// TIA Portal V17 export
// export: Created 2023-04-11T09:33:28.1593293Z, ExportSetting WithDefaults, DisplayName Totally Integrated Automation Portal, DisplayVersion V17 Update 3, DisplayName TIA Portal Openness, DisplayVersion V17 Update 3, DisplayName TIA Portal Version Control Interface, DisplayVersion V17, DisplayName SINAMICS Startdrive Advanced, DisplayVersion V17 Update2, DisplayName SINAMICS Startdrive G130, G150, S120, S150, SINAMICS MV, S210, DisplayVersion V17 Update2, DisplayName SINAMICS Startdrive G110M, G120, G120C, G120D, G120P, G115D, DisplayVersion V17 Update2, DisplayName STEP 7 Professional, DisplayVersion V17 Update 3, DisplayName STEP 7 Safety, DisplayVersion V17, DisplayName WinCC UA Professional, DisplayVersion V17 Update 3
FUNCTION_BLOCK "FB_stdCylinder"   // FB121, LAD
TITLE = Standart cylinder control
{ S7_Optimized_Access := 'TRUE' }
VERSION : 0.1
// stored: AutoNumber true, IsIECCheckEnabled false, IsRetainMemResEnabled false, MemoryReserve 100, SetENOAutomatically false, UDAEnableTagReadback false
   VAR_INPUT
      Double_Coil : Bool;
      Request_A : Bool;
      Request_B : Bool;
      Sensor_A : Bool;
      With_A : Bool;
      Sensor_B : Bool;
      With_B : Bool;
      Enable_A : Bool;
      Enable_B : Bool;
      Monitoring_On : Bool;
      SensorDelay_A : Time;
      SensorDelay_B : Time;
      TimeForError_A : Time;
      TimeForError_B : Time;
   END_VAR
   VAR_OUTPUT
      Out_A : Bool;
      Out_B : Bool;
      Done_A : Bool;
      Done_B : Bool;
      Error_A : Bool;
      Error_B : Bool;
      Error_moveBlock : Bool;
   END_VAR
   VAR
      FB_FaultModule_Instance { S7_SetPoint := 'True'} : "FB_faultModule";
      IEC_Timer_0_Instance { S7_SetPoint := 'True'} : TON_TIME;
      IEC_Timer_0_Instance_1 { S7_SetPoint := 'True'} : TON_TIME;
      IEC_Timer_0_Instance_2 { S7_SetPoint := 'True'} : TON_TIME;
      IEC_Timer_0_Instance_3 { S7_SetPoint := 'True'} : TON_TIME;
   END_VAR
   VAR_TEMP
      Out_A_temp : Bool;
      Out_B_temp : Bool;
   END_VAR
BEGIN

REGION Network 1: OUT A
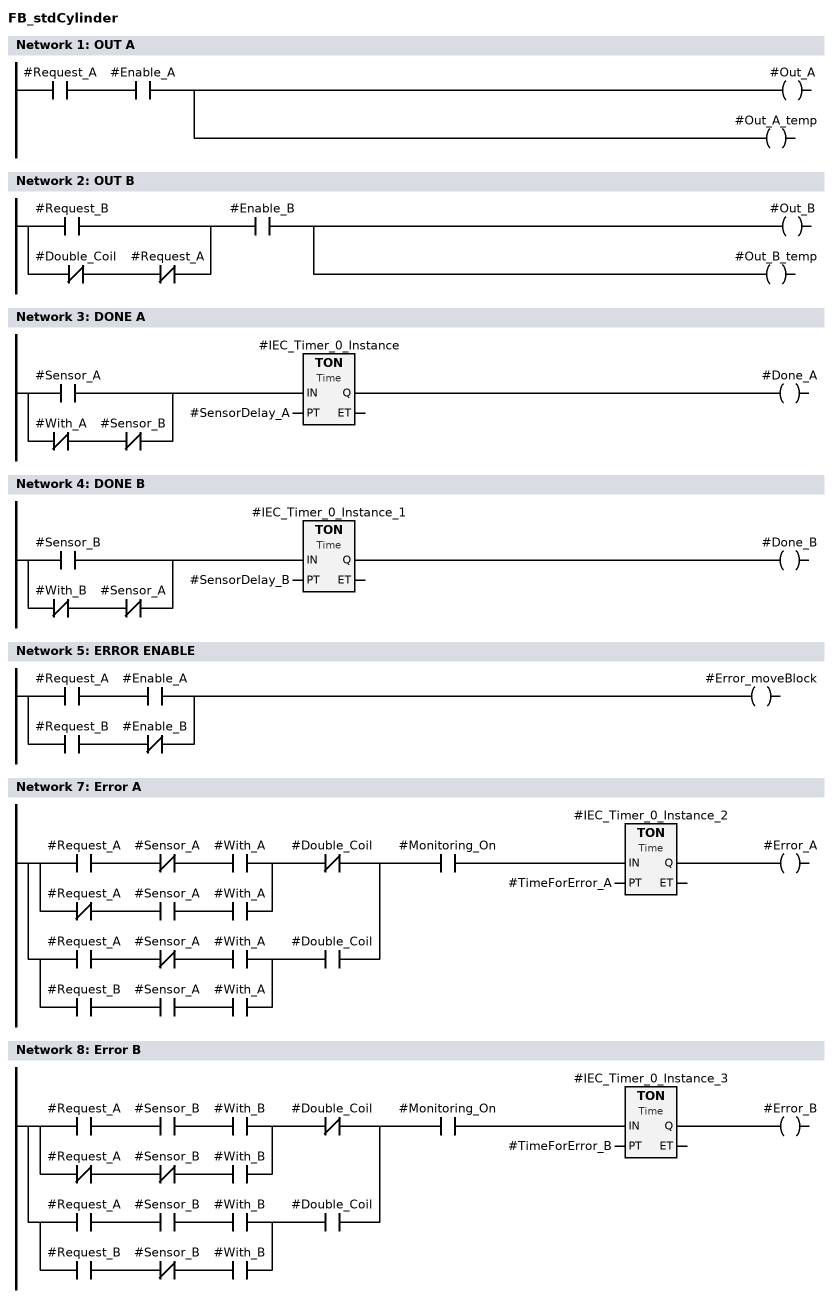
   RUNG wire#powerrail
      Contact( #Request_A )
      Contact( #Enable_A )
      wire#w1
      Coil( #Out_A )
   END_RUNG
   RUNG wire#w1
      Coil( #Out_A_temp )
   END_RUNG
   // the same network as SCL:
   #Out_A := #Request_A AND #Enable_A;
   #Out_A_temp := #Out_A;
END_REGION

REGION Network 2: OUT B
   RUNG wire#powerrail
      Contact( #Request_B )
      wire#w1
      Contact( #Enable_B )
      wire#w2
      Coil( #Out_B )
   END_RUNG
   RUNG wire#powerrail
      I_Contact( #Double_Coil )
      I_Contact( #Request_A )
   END_RUNG wire#w1
   RUNG wire#w2
      Coil( #Out_B_temp )
   END_RUNG
   // the same network as SCL:
   #Out_B := (#Request_B OR (NOT #Double_Coil AND NOT #Request_A)) AND #Enable_B;
   #Out_B_temp := #Out_B;
END_REGION

REGION Network 3: DONE A
   RUNG wire#powerrail
      Contact( #Sensor_A )
      wire#w1
      { S7_Templates := "time_type := Time" } #IEC_Timer_0_Instance.TON(pt := #SensorDelay_A, et =>)
      Coil( #Done_A )
   END_RUNG
   RUNG wire#powerrail
      I_Contact( #With_A )
      I_Contact( #Sensor_B )
   END_RUNG wire#w1
   // the same network as SCL:
   #IEC_Timer_0_Instance(IN := #Sensor_A OR (NOT #With_A AND NOT #Sensor_B), PT := #SensorDelay_A);   // TON
   #Done_A := #IEC_Timer_0_Instance.Q;
END_REGION

REGION Network 4: DONE B
   RUNG wire#powerrail
      Contact( #Sensor_B )
      wire#w1
      { S7_Templates := "time_type := Time" } #IEC_Timer_0_Instance_1.TON(pt := #SensorDelay_B, et =>)
      Coil( #Done_B )
   END_RUNG
   RUNG wire#powerrail
      I_Contact( #With_B )
      I_Contact( #Sensor_A )
   END_RUNG wire#w1
   // the same network as SCL:
   #IEC_Timer_0_Instance_1(IN := #Sensor_B OR (NOT #With_B AND NOT #Sensor_A), PT := #SensorDelay_B);   // TON
   #Done_B := #IEC_Timer_0_Instance_1.Q;
END_REGION

REGION Network 5: ERROR ENABLE
   RUNG wire#powerrail
      Contact( #Request_A )
      Contact( #Enable_A )
      wire#w1
      Coil( #Error_moveBlock )
   END_RUNG
   RUNG wire#powerrail
      Contact( #Request_B )
      I_Contact( #Enable_B )
   END_RUNG wire#w1
   // the same network as SCL:
   #Error_moveBlock := (#Request_A AND #Enable_A) OR (#Request_B AND NOT #Enable_B);
END_REGION

REGION Network 7: Error A
   RUNG wire#powerrail
      Contact( #Request_A )
      I_Contact( #Sensor_A )
      Contact( #With_A )
      wire#w1
      I_Contact( #Double_Coil )
      wire#w2
      Contact( #Monitoring_On )
      { S7_Templates := "time_type := Time" } #IEC_Timer_0_Instance_2.TON(pt := #TimeForError_A, et =>)
      Coil( #Error_A )
   END_RUNG
   RUNG wire#powerrail
      I_Contact( #Request_A )
      Contact( #Sensor_A )
      Contact( #With_A )
   END_RUNG wire#w1
   RUNG wire#powerrail
      Contact( #Request_A )
      I_Contact( #Sensor_A )
      Contact( #With_A )
      wire#w3
      Contact( #Double_Coil )
   END_RUNG wire#w2
   RUNG wire#powerrail
      Contact( #Request_B )
      Contact( #Sensor_A )
      Contact( #With_A )
   END_RUNG wire#w3
   // the same network as SCL:
   #IEC_Timer_0_Instance_2(IN := ((((#Request_A AND NOT #Sensor_A AND #With_A) OR (NOT #Request_A AND #Sensor_A AND #With_A)) AND NOT #Double_Coil) OR (((#Request_A AND NOT #Sensor_A AND #With_A) OR (#Request_B AND #Sensor_A AND #With_A)) AND #Double_Coil)) AND #Monitoring_On,   // TON
                           PT := #TimeForError_A);
   #Error_A := #IEC_Timer_0_Instance_2.Q;
END_REGION

REGION Network 8: Error B
   RUNG wire#powerrail
      Contact( #Request_A )
      Contact( #Sensor_B )
      Contact( #With_B )
      wire#w1
      I_Contact( #Double_Coil )
      wire#w2
      Contact( #Monitoring_On )
      { S7_Templates := "time_type := Time" } #IEC_Timer_0_Instance_3.TON(pt := #TimeForError_B, et =>)
      Coil( #Error_B )
   END_RUNG
   RUNG wire#powerrail
      I_Contact( #Request_A )
      I_Contact( #Sensor_B )
      Contact( #With_B )
   END_RUNG wire#w1
   RUNG wire#powerrail
      Contact( #Request_A )
      Contact( #Sensor_B )
      Contact( #With_B )
      wire#w3
      Contact( #Double_Coil )
   END_RUNG wire#w2
   RUNG wire#powerrail
      Contact( #Request_B )
      I_Contact( #Sensor_B )
      Contact( #With_B )
   END_RUNG wire#w3
   // the same network as SCL:
   #IEC_Timer_0_Instance_3(IN := ((((#Request_A AND #Sensor_B AND #With_B) OR (NOT #Request_A AND NOT #Sensor_B AND #With_B)) AND NOT #Double_Coil) OR (((#Request_A AND #Sensor_B AND #With_B) OR (#Request_B AND NOT #Sensor_B AND #With_B)) AND #Double_Coil)) AND #Monitoring_On,   // TON
                           PT := #TimeForError_B);
   #Error_B := #IEC_Timer_0_Instance_3.Q;
END_REGION
END_FUNCTION_BLOCK
